PROGRAM MAIN
VAR
	fbDev1	:	FB_ExampleDeviceSM_All;
	fbDev2	:	FB_ExampleDeviceSM_All;
	
	rtInit	:	R_TRIG;
	Initialize	:	BOOL := TRUE;
	
	DemoMode: BOOL :=TRUE;
	fbDev3	:	FB_ExampleDeviceSM_DB;

END_VAR

//Sub-system Device PLC

IF DemoMode	THEN

//Fast Faults must run first
Fast_Faults();

IF Initialize THEN
	fbDev1(cBase := 10,
		fbFastFaultOutput := g_FastFaultOutput1,
		fbArbiter := g_fbArbiter);
	fbDev2(cBase := 1000,
		fbFastFaultOutput := g_FastFaultOutput1,
		fbArbiter := g_fbArbiter);
	g_fbArbiter.A_Init();

	fbDev3(cBase := 0,iDBID:=1,sDBNetId:='172.21.42.53.1.1',sDeviceID:='1',
		fbArbiter := g_fbArbiter,
		fbFastFaultOutput := g_FastFaultOutput1);
	Initialize := FALSE;
END_IF

//Example devices
fbDev1(fbFastFaultOutput := g_FastFaultOutput1,
		fbArbiter := g_fbArbiter);
fbDev2(fbFastFaultOutput := g_FastFaultOutput1,
		fbArbiter := g_fbArbiter);


fbDev3(fbArbiter := g_fbArbiter,
		fbFastFaultOutput := g_FastFaultOutput1);
		

		
PMPS_Arbiter();

Fast_Faults_Evaluate();

MachineSimulation();

ELSE
	TestSetups();
END_IF

ACTION FB_Vis:
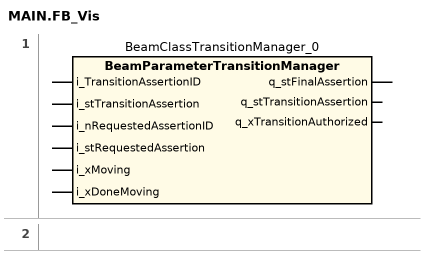
// NETWORK 1
BeamClassTransitionManager_0(); // BeamParameterTransitionManager

// NETWORK 2
END_ACTION

ACTION Initialize:

END_ACTION

END_PROGRAM

(* stored: Version 1.1.0.1, ProductVersion 3.1.4022.12
   POU MAIN: Id {8a7bcfd2-1a2b-4363-aa47-c19391bf1f9c}, SpecialFunc None
   Action FB_Vis: Id {dbfecf7e-be1a-0abd-04cf-64b55d658bf1}
   Action Initialize: Id {b0ee480a-3d4b-001d-04c4-43cdc47895c8} *)
